{attribute 'GeneratedUsingTerminal: EL6690-0001-0000'}
{attribute addProperty BoxType "EL6690-0001-0000"}
{attribute addProperty Id "StatusAT %I*Status_D30DC33F1InputsEMPTY_STRUCTURE0OutputsEMPTY_STRUCTURE0WcStateAT %I*WcState_9091E0EB2InfoDataAT %I*InfoData_94A18F5E2"}
{attribute addProperty CRC "1566795143"}
{attribute addProperty Size "5"}
TYPE EL6690_5D636587 EXTENDS EtcSlaveTerminalBase_947E5A46 :
STRUCT
	{attribute addProperty Name "Status"}
	Status : Status_D30DC33F;
	{attribute addProperty Name "Inputs"}
	Inputs : EMPTY_STRUCTURE;
	{attribute addProperty Name "Outputs"}
	Outputs : EMPTY_STRUCTURE;
	{attribute addProperty Name "WcState"}
	WcState : WcState_9091E0EB;
	{attribute addProperty Name "InfoData"}
	InfoData : InfoData_94A18F5E;
END_STRUCT
END_TYPE

(* stored: Version 1.2.0.0, ProductVersion 3.1.4024.9
   DUT EL6690_5D636587: Id {7489249a-c6be-4944-8d68-fe22f0f34262} *)
